# EPICS StreamDevice protocol: streamdeviceApp/Db/RC3U-1.proto
Terminator = CR;

#Read Alarm State Level 1
ReadAlarmLevel1 {out ".0118rAlrmLv1%0<sum8>"; in "#01180rAlrmLv1%1d%(\$1)1d%(\$2)1d%(\$3)1d%(\$4)1d%(\$5)1d%0<sum8>";}

#Read Alarm State Level 2
ReadAlarmLevel21 {out ".0119rAlrmLv21%0<sum8>"; in "#01190rAlrmLv21%1d%(\$1)1d%(\$2)1d%(\$3)1d%(\$4)1d%(\$5)1d%(\$6)1d%(\$7)1d%0<sum8>";}
ReadAlarmLevel22 {out ".0119rAlrmLv22%0<sum8>"; in "#01190rAlrmLv22%1d%(\$1)1d%(\$2)1d%(\$3)1d%(\$4)1d%(\$5)1d%(\$6)1d%(\$7)1d%0<sum8>";}
